// TwinCAT 3 PLC project CNM_CycleManager
// Title: CNM_CycleManager
// Company: ekvip automation GmbH
// Author: tdie
// ProjectVersion: 0.1.1.0
// Description: A library to provide Cycle management for use in simple state machines. .. <legal notes> legal notes ================= | SPDX-FileCopyrightText: © 2024 ekvip automation GmbH <info@ekvip.de> | SPDX-License-Identifier: Apache-2.0 | For details check: Apache-2.0_ .. _Apache-2.0: https://www.apache.org/licenses/LICENSE-2.0 .. </legal notes>
// ProgramVersion: 3.1.4026.19
// libraries:
//   CNM_AbstractObject, * (ekvip automation GmbH)
//   CNM_AssertionInterfaces, * (ekvip automation GmbH)
//   CNM_CommandInterfaces, * (ekvip automation GmbH)
//   CNM_CycleManagerInterfaces, * (ekvip automation GmbH)
//   CNM_MessageInterfaces, * (ekvip automation GmbH)
//   CNM_ReturnTypes, * (ekvip automation GmbH)
//   Tc2_Standard, * (Beckhoff Automation GmbH)
//   Tc2_System, * (Beckhoff Automation GmbH)
// project tree:
//   Commands/classes/ WaitCommand.TcPOU
//   Configurators/classes/ CycleManagerConfigurator.TcPOU, CycleManagerDefaultConfigurator.TcPOU, CycleManagerDefaultPausing.TcPOU, CycleManagerDefaultStepping.TcPOU, CycleManagerStepConfigurator.TcPOU, CycleManagerStepPausing.TcPOU, CycleManagerStepStepping.TcPOU
//   CycleManager/classes/ AbstractCycleManager.TcPOU, SimpleCycleManager.TcPOU
//   CycleManager/interfaces/ ICycleManagerStepParameters.TcIO
//   Project Information/ F_GetCompany.TcPOU, F_GetTitle.TcPOU, F_GetVersion.TcPOU
//   Version/ Global_Version.TcGVL

// ---- Version/Global_Version.TcGVL
{attribute 'TcGenerated'}
{attribute 'no-analysis'}
{attribute 'linkalways'}
// This function has been automatically generated from the project information.
VAR_GLOBAL CONSTANT
	{attribute 'const_non_replaced'}
	stLibVersion_CNM_CycleManager : ST_LibVersion := (iMajor := 0, iMinor := 1, iBuild := 1, iRevision := 0, nFlags := 0, sVersion := '0.1.1.0');
END_VAR

// ---- CycleManager/interfaces/ICycleManagerStepParameters.TcIO
(*

## Short summary
An interface to provide configurations for cycle manager steps.
Used internally to allow better fluent implementation.

.. <legal notes>

legal notes
=================
| SPDX-FileCopyrightText: © 2024 ekvip automation GmbH <info@ekvip.de>
| SPDX-License-Identifier: Apache-2.0
| For details check: Apache-2.0_

.. _Apache-2.0: https://www.apache.org/licenses/LICENSE-2.0

.. </legal notes>



*)
INTERFACE INTERNAL ICycleManagerStepParameters EXTENDS __System.IQueryInterface

PROPERTY currentErrorStep : DINT
SET
END_SET
END_PROPERTY

PROPERTY currentPauseEnabled : BOOL
SET
END_SET
END_PROPERTY

PROPERTY currentSteppingEnabled : BOOL
SET
END_SET
END_PROPERTY

PROPERTY currentStepWidth : DINT
SET
END_SET
END_PROPERTY

PROPERTY currentStopRequestMode :CNM_CycleManagerInterfaces.StepStopRequestMode
SET
END_SET
END_PROPERTY

PROPERTY currentTimeout : TIME
SET
END_SET
END_PROPERTY

PROPERTY currentTimeoutStep : DINT
SET
END_SET
END_PROPERTY

END_INTERFACE

// ---- Commands/classes/WaitCommand.TcPOU
(*

## Short summary
A simple command to wait for a given time.

.. <legal notes>

legal notes
=================
| SPDX-FileCopyrightText: © 2024 ekvip automation GmbH <info@ekvip.de>
| SPDX-License-Identifier: Apache-2.0
| For details check: Apache-2.0_

.. _Apache-2.0: https://www.apache.org/licenses/LICENSE-2.0

.. </legal notes>

*)
FUNCTION_BLOCK FINAL WaitCommand EXTENDS CNM_AbstractObject.Object IMPLEMENTS CNM_CommandInterfaces.ICommand
VAR
	timeToWait :TIME;
	timer :TON;
END_VAR

(*

## Short summary
This abstract property returns the class name of the concrete object, 
which is useful for logging/debugging purpose or to check the class name
for ``__DELETE`` in factories (sometimes it's necessary to do more 
than just to free the memory).

.. <legal notes>

legal notes
=================
| SPDX-FileCopyrightText: © 2022 ekvip automation GmbH <info@ekvip.de>
| SPDX-License-Identifier: Apache-2.0
| For details check: Apache-2.0_

.. _Apache-2.0: https://www.apache.org/licenses/LICENSE-2.0

.. </legal notes>

*)
PROPERTY className : CNM_AbstractObject.ClassName
GET
className := 'CNM_CycleManager.WaitCommand';
END_GET
END_PROPERTY

(*

## Short summary
Executes the action associated with this command.

.. <legal notes>

legal notes
=================
| SPDX-FileCopyrightText: © 2022 ekvip automation GmbH <info@ekvip.de>
| SPDX-License-Identifier: Apache-2.0
| For details check: Apache-2.0_

.. _Apache-2.0: https://www.apache.org/licenses/LICENSE-2.0

.. </legal notes>

*)
METHOD executeCommand : CNM_ReturnTypes.SingleExecutionState
VAR_INPUT
	(*control bit to start or abort the command*)
	execute	: BOOL;
END_VAR
THIS^.timer(IN := execute AND (THIS^.waitTime <> T#0S), PT := THIS^.waitTime);
IF(THIS^.timer.Q OR_ELSE THIS^.waitTime = T#0S)THEN
	executeCommand := CNM_ReturnTypes.SingleExecutionState.SUCCESS;
ELSE
	executeCommand := CNM_ReturnTypes.SingleExecutionState.BUSY;	
END_IF
END_METHOD

(*

## Short summary
The constructor ``FB_init`` is needed to create an unique hash code.
The hash code is a pseudo random number create with a xorshift_ algorithm.
It can be overwritten on derivations, because it will be called implicit, ``SUPER^.FB_init()`` is not required.
For more information check: `Behavoir with derived function blocks`_

.. _Behavoir with derived function blocks: https://infosys.beckhoff.com/content/1033/tc3_plc_intro/5482088715.html?id=6983869892358031022
.. _xorshift: https://en.wikipedia.org/wiki/Xorshift

.. <legal notes>

legal notes
=================
| SPDX-FileCopyrightText: © 2022 ekvip automation GmbH <info@ekvip.de>
| SPDX-License-Identifier: Apache-2.0
| For details check: Apache-2.0_

.. _Apache-2.0: https://www.apache.org/licenses/LICENSE-2.0

.. </legal notes>

*)
METHOD FB_init :BOOL
VAR_INPUT
	(* if TRUE, the retain variables are initialized (warm start / cold start)*)
	bInitRetains	:BOOL;
	(* if TRUE, the instance afterwards gets moved into the copy code (online change) *)
	bInCopyCode	:BOOL;
	(* time to wait until return state is success *)
	waitTime :TIME;
END_VAR
THIS^.timeToWait := waitTime;
END_METHOD

(*

## Short summary
This property sets or gets the time to wait for until the command returns SUCCESS.

.. <legal notes>

legal notes
=================
| SPDX-FileCopyrightText: © 2022 ekvip automation GmbH <info@ekvip.de>
| SPDX-License-Identifier: Apache-2.0
| For details check: Apache-2.0_

.. _Apache-2.0: https://www.apache.org/licenses/LICENSE-2.0

.. </legal notes>

*)
PROPERTY waitTime : TIME
GET
waitTime := THIS^.timeToWait;
END_GET
SET
THIS^.timeToWait := waitTime;
END_SET
END_PROPERTY

END_FUNCTION_BLOCK

// ---- Configurators/classes/CycleManagerConfigurator.TcPOU
(*

## Short summary
A class to provide fluent access to the configuration scope of a cycle manager.

.. <legal notes>

legal notes
=================
| SPDX-FileCopyrightText: © 2024 ekvip automation GmbH <info@ekvip.de>
| SPDX-License-Identifier: Apache-2.0
| For details check: Apache-2.0_

.. _Apache-2.0: https://www.apache.org/licenses/LICENSE-2.0

.. </legal notes>



*)
FUNCTION_BLOCK INTERNAL CycleManagerConfigurator IMPLEMENTS CNM_CycleManagerInterfaces.ICycleManagerConfigurationScope
VAR
	cycleManagerDefault :CNM_CycleManagerInterfaces.ICycleManagerDefaultParameters;
	cycleManagerStep :ICycleManagerStepParameters;
	stepConfigurator :CycleManagerStepConfigurator();
	defaultConfigurator :CycleManagerDefaultConfigurator();
END_VAR

(*

## Short summary
Initializes the CycleManagerConfigurator with required cycle manager parameters.

.. <legal notes>

legal notes
=================
| SPDX-FileCopyrightText: © 2025 ekvip automation GmbH <info@ekvip.de>
| SPDX-License-Identifier: Apache-2.0
| For details check: Apache-2.0_

.. _Apache-2.0: https://www.apache.org/licenses/LICENSE-2.0

.. </legal notes>

*)
//FB_Init is always available implicitly and it is used primarily for initialization.
//The return value is not evaluated. For a specific influence, you can also declare the
//methods explicitly and provide additional code there with the standard initialization
//code. You can evaluate the return value.
METHOD FB_Init: BOOL
VAR_INPUT
    bInitRetains: BOOL; // TRUE: the retain variables are initialized (reset warm / reset cold)
    bInCopyCode: BOOL;  // TRUE: the instance will be copied to the copy code afterward (online change)   
	cycleManagerDefault :CNM_CycleManagerInterfaces.ICycleManagerDefaultParameters; //Interface for default cycle manager parameters
	cycleManagerStep :ICycleManagerStepParameters; //Interface for step-specific cycle manager parameters
END_VAR
THIS^.cycleManagerDefault := cycleManagerDefault;
THIS^.cycleManagerStep := cycleManagerStep;
THIS^.defaultConfigurator.cycleManager := cycleManagerDefault;
THIS^.stepConfigurator.cycleManager := cycleManagerStep;
END_METHOD

(*

## Short summary
Provides access to sequence-level configuration for all cycle manager steps.

### Purpose and usage
This property returns the sequence configuration interface that allows setting default parameters
for all steps in the cycle manager. It provides a fluent interface for configuring sequence-wide
settings that apply to the entire cycle execution.

The sequence configuration affects all steps uniformly and provides default values for:
- Pause behavior
- Stepping mode settings
- Stop request handling
- Other sequence-wide parameters


### typical usage patterns
1. **Setting default timeouts**: Configure default timeout for all steps
2. **Pause configuration**: Set pause behavior for the entire sequence
3. **Stepping mode**: Configure stepping mode defaults
4. **Stop handling**: Define how stop requests are handled globally

### When to use
- When you need to configure default behavior for all steps
- To set sequence-wide parameters that apply uniformly
- For configuring global cycle manager behavior
- When implementing consistent behavior across all steps

### Example
```
// Configure sequence defaults
cycleManager.configuration.configuration.sequence
    .pauseConfiguration
        .pauseAllowed(TRUE)
        .pauseTimeout(T#5S);

// Set stepping mode for entire sequence
cycleManager.configuration.configuration.sequence
    .steppingConfiguration
        .steppingEnabled(debugMode)
        .autoStepDelay(T#100MS);

// Configure stop request handling
cycleManager.configuration.configuration.sequence
    .stopRequestConfiguration
        .stopAllowed(TRUE)
        .immediateStop(FALSE);

```
.. <legal notes>

legal notes
=================
| SPDX-FileCopyrightText: © 2025 ekvip automation GmbH <info@ekvip.de>
| SPDX-License-Identifier: Apache-2.0
| For details check: Apache-2.0_

.. _Apache-2.0: https://www.apache.org/licenses/LICENSE-2.0

.. </legal notes>

*)
PROPERTY sequence : CNM_CycleManagerInterfaces.ISequenceConfiguration
GET
sequence := defaultConfigurator;
END_GET
END_PROPERTY

(*

## Short summary
Provides access to step-specific configuration for individual cycle manager steps.

### Purpose and usage
This property returns the step configuration interface that allows setting parameters
for specific steps in the cycle manager. It provides a fluent interface for configuring
individual step behavior that overrides the sequence defaults.

The step configuration allows fine-grained control over individual steps including:
- Step-specific timeouts
- Individual pause behavior
- Custom stepping settings
- Step-specific stop handling

### typical usage patterns
1. **Step-specific timeouts**: Override default timeout for critical steps
2. **Disable pause**: Prevent pausing on critical operation steps
3. **Skip stepping**: Make certain steps non-steppable in debug mode
4. **Custom behavior**: Define unique behavior for specific steps

### When to use
- When specific steps need different behavior than the sequence default
- For critical steps that should not be pausable or steppable
- To set custom timeouts for long-running operations
- When implementing step-specific error handling

### Example
```
// Configure specific step with custom timeout
cycleManager.configuration.configuration.step
    .forStep(MySteps.LONG_OPERATION)
    .setTimeout(T#30S)
    .pauseAllowed(FALSE);  // Critical step - no pause allowed

// Configure multiple steps
cycleManager.configuration.configuration.step
    .forStep(MySteps.INIT)
    .setTimeout(T#5S)
    .steppingAllowed(TRUE);

cycleManager.configuration.configuration.step
    .forStep(MySteps.CRITICAL_PROCESS)
    .setTimeout(T#10S)
    .pauseAllowed(FALSE)
    .stopAllowed(FALSE);  // Must complete once started

// Configure error step
cycleManager.configuration.configuration.step
    .forStep(DefaultSteps.STEP.ERROR)
    .setTimeout(T#0S)  // No timeout in error state
    .steppingAllowed(TRUE);  // Allow stepping through error handling
```

.. <legal notes>

legal notes
=================
| SPDX-FileCopyrightText: © 2025 ekvip automation GmbH <info@ekvip.de>
| SPDX-License-Identifier: Apache-2.0
| For details check: Apache-2.0_

.. _Apache-2.0: https://www.apache.org/licenses/LICENSE-2.0

.. </legal notes>


*)
PROPERTY step : CNM_CycleManagerInterfaces.IStepConfiguration
GET
VAR_INST
	conf :CycleManagerStepConfigurator();
END_VAR
step := stepConfigurator;
END_GET
END_PROPERTY

END_FUNCTION_BLOCK

// ---- Configurators/classes/CycleManagerStepConfigurator.TcPOU
(*

## Short summary
A class to provide fluent access to the current step configuration of a cycle manager.

.. <legal notes>

legal notes
=================
| SPDX-FileCopyrightText: © 2024 ekvip automation GmbH <info@ekvip.de>
| SPDX-License-Identifier: Apache-2.0
| For details check: Apache-2.0_

.. _Apache-2.0: https://www.apache.org/licenses/LICENSE-2.0

.. </legal notes>



*)
FUNCTION_BLOCK INTERNAL CycleManagerStepConfigurator IMPLEMENTS CNM_CycleManagerInterfaces.IStepConfiguration, CNM_CycleManagerInterfaces.IStopRequestConfiguration
VAR
	parameters :ICycleManagerStepParameters;
	pauserator :CycleManagerStepPausing();
	steperator :CycleManagerStepStepping();
END_VAR

(*

## Short summary
Sets the stop request behavior to execute after successful step completion for the current step.

### Purpose and usage
This method configures the current step to process stop requests only after the step has completed successfully.
This setting overrides the sequence default for this specific step. When this mode is active, stop requests
received during step execution will be deferred until the step completes with success.

This ensures that the specific step completes successfully before the cycle is stopped,
maintaining data integrity and process consistency for critical operations.

### typical usage patterns
1. **Critical steps**: Ensure specific steps complete before stopping
2. **Transaction steps**: Finish data transactions cleanly
3. **Safety operations**: Complete safety-critical steps
4. **Production steps**: Avoid partial operations on key steps

### When to use
- For steps that must complete successfully before stopping
- When specific operations should not be interrupted
- For data consistency in critical steps
- To override sequence defaults for important steps

### Example
```
// Configure specific step for safe stopping
cycleManager.configuration.configuration.step
    .stopRequest
    .afterSuccess();

// Apply to critical step during configuration
CASE cycleManager.steps.current OF
    MySteps.INIT:
        // Configure next critical step
        cycleManager.configuration.configuration.step
            .timeout := T#10S;
        cycleManager.configuration.configuration.step
            .stopRequest.afterSuccess();
        cycleManager.steps.next := MySteps.CRITICAL_WRITE;
        
    MySteps.CRITICAL_WRITE:
        // This step will complete before stop is processed
        IF writeCriticalData() THEN
            cycleManager.steps.next := MySteps.NEXT_STEP;
        END_IF;
END_CASE
```


.. <legal notes>

legal notes
=================
| SPDX-FileCopyrightText: © 2025 ekvip automation GmbH <info@ekvip.de>
| SPDX-License-Identifier: Apache-2.0
| For details check: Apache-2.0_

.. _Apache-2.0: https://www.apache.org/licenses/LICENSE-2.0

.. </legal notes>

*)
METHOD afterSuccessfulStep
THIS^.cycleManager.currentStopRequestMode := CNM_CycleManagerInterfaces.StepStopRequestMode.AFTER_SUCCESSFUL_STEP;
END_METHOD

(*

## Short summary
Gets or sets the cycle manager step parameters interface used by this configurator.

### Purpose and usage
This property provides access to the underlying cycle manager step parameters interface.
It allows getting the current cycle manager instance and setting a new one if needed.

When setting a new cycle manager, all internal configurators (stepping and pausing)
are automatically updated to use the new instance. This property manages step-specific
parameters that override sequence defaults.

### typical usage patterns
1. **Initialization**: Set during configurator creation
2. **Runtime changes**: Switch cycle manager instances
3. **Access parameters**: Get current cycle manager for direct access
4. **Step-specific config**: Access step-level parameters

### When to use
- During initialization to set the cycle manager
- When switching between different cycle manager implementations
- For direct access to step-specific parameters
- In factory patterns for dynamic configuration

### Example
```
// Get current cycle manager
VAR
    currentManager : ICycleManagerStepParameters;
END_VAR

currentManager := stepConfigurator.cycleManager;

// Set new cycle manager
VAR
    newManager : MyCycleManagerStepImplementation;
END_VAR

stepConfigurator.cycleManager := newManager;
// All sub-configurators now use newManager

// Direct parameter access
IF stepConfigurator.cycleManager.currentTimeout > T#5S THEN
    // Handle long timeout for current step
END_IF;
```

.. <legal notes>

legal notes
=================
| SPDX-FileCopyrightText: © 2025 ekvip automation GmbH <info@ekvip.de>
| SPDX-License-Identifier: Apache-2.0
| For details check: Apache-2.0_

.. _Apache-2.0: https://www.apache.org/licenses/LICENSE-2.0

.. </legal notes>


*)
PROPERTY cycleManager : ICycleManagerStepParameters
GET
cycleManager := THIS^.parameters;
END_GET
SET
THIS^.parameters := cycleManager;
THIS^.steperator.cycleManager := THIS^.cycleManager;
THIS^.pauserator.cycleManager := THIS^.cycleManager;
END_SET
END_PROPERTY

(*

## Short summary
This property sets the next step in case of an error.
Is reset to the default ERROR_STEP when the current step changes.

.. <legal notes>

legal notes
=================
| SPDX-FileCopyrightText: © 2024 ekvip automation GmbH <info@ekvip.de>
| SPDX-License-Identifier: Apache-2.0
| For details check: Apache-2.0_

.. _Apache-2.0: https://www.apache.org/licenses/LICENSE-2.0

.. </legal notes>

*)
PROPERTY errorStep : DINT
SET
THIS^.cycleManager.currentErrorStep := errorStep;
END_SET
END_PROPERTY

(*

## Short summary
Initializes the CycleManagerStepConfigurator and its sub-configurators.

.. <legal notes>

legal notes
=================
| SPDX-FileCopyrightText: © 2025 ekvip automation GmbH <info@ekvip.de>
| SPDX-License-Identifier: Apache-2.0
| For details check: Apache-2.0_

.. _Apache-2.0: https://www.apache.org/licenses/LICENSE-2.0

.. </legal notes>

*)
//FB_Init is always available implicitly and it is used primarily for initialization.
//The return value is not evaluated. For a specific influence, you can also declare the
//methods explicitly and provide additional code there with the standard initialization
//code. You can evaluate the return value.
METHOD FB_Init: BOOL
VAR_INPUT
    bInitRetains: BOOL; // TRUE: the retain variables are initialized (reset warm / reset cold)
    bInCopyCode: BOOL;  // TRUE: the instance will be copied to the copy code afterward (online change)   
END_VAR
THIS^.steperator.cycleManager := THIS^.cycleManager;
THIS^.pauserator.cycleManager := THIS^.cycleManager;
END_METHOD

(*

## Short summary
Sets the stop request behavior to ignore all stop requests for the current step.

### Purpose and usage
This method configures the current step to completely ignore all stop requests.
This setting overrides the sequence default for this specific step. When this mode
is active, stop requests will not be processed at all during this step, and the
step will continue running until completion or error.

This mode should be used with extreme caution as it prevents normal stopping
mechanisms from working for the specific step.

### typical usage patterns
1. **Atomic operations**: Steps that must complete without interruption
2. **Safety sequences**: Emergency procedures for specific steps
3. **Critical writes**: Database or file operations that cannot be stopped
4. **Hardware operations**: Steps controlling physical processes

### When to use
- For step-specific critical operations that must complete
- During safety-critical step sequences
- For atomic operations within a larger sequence
- When a specific step must ignore stop requests
- Use with extreme caution - limits operator control

### Example
```
// Configure specific step to ignore stops
cycleManager.configuration.configuration.step
    .stopRequest
    .ignore();

// Apply to critical hardware operation
CASE cycleManager.steps.current OF
    MySteps.PREPARE_CRITICAL:
        // Configure next step to ignore stops
        cycleManager.configuration.configuration.step
            .stopRequest.ignore();
        cycleManager.steps.next := MySteps.CRITICAL_HARDWARE_OP;
        
    MySteps.CRITICAL_HARDWARE_OP:
        // This step ignores all stop requests
        IF performCriticalHardwareOperation() THEN
            // Re-enable stop handling for next step
            cycleManager.configuration.configuration.step
                .stopRequest.afterSuccess();
            cycleManager.steps.next := MySteps.NORMAL_OPERATION;
        END_IF;
END_CASE

// Stop requests during critical step will be ignored
IF stopButton THEN
    cycleManager.requestStop();  // No effect on CRITICAL_HARDWARE_OP
END_IF;
```

.. <legal notes>

legal notes
=================
| SPDX-FileCopyrightText: © 2025 ekvip automation GmbH <info@ekvip.de>
| SPDX-License-Identifier: Apache-2.0
| For details check: Apache-2.0_

.. _Apache-2.0: https://www.apache.org/licenses/LICENSE-2.0

.. </legal notes>


*)
METHOD ignore
THIS^.cycleManager.currentStopRequestMode := CNM_CycleManagerInterfaces.StepStopRequestMode.IGNORE;
END_METHOD

(*

## Short summary
Sets the stop request behavior to always process stop requests immediately for the current step.

### Purpose and usage
This method configures the current step to always process stop requests immediately,
regardless of the step's execution state or outcome. This setting overrides the sequence
default for this specific step. Stop requests are handled as soon as they are received,
potentially interrupting the current operation.

This mode provides the most responsive stop behavior for the specific step but may
interrupt operations that are in progress.

### typical usage patterns
1. **Non-critical steps**: Allow immediate stop on safe steps
2. **Wait steps**: Enable quick response during waits
3. **User interaction**: Responsive stops during user steps
4. **Idle states**: Allow immediate stop when idle

### When to use
- For steps where immediate stop response is acceptable
- During wait or idle steps
- For non-critical operations that can be interrupted
- To override restrictive sequence defaults for specific steps

### Example
```
// Configure specific step for immediate stop
cycleManager.configuration.configuration.step
    .stopRequest
    .always();

// Apply to wait steps
CASE cycleManager.steps.current OF
    MySteps.WAIT_FOR_INPUT:
        // This step can be interrupted immediately
        cycleManager.configuration.configuration.step
            .stopRequest.always();
        IF inputReceived THEN
            cycleManager.steps.next := MySteps.PROCESS_INPUT;
        END_IF;
        
    MySteps.IDLE:
        // Idle step allows immediate stop
        cycleManager.configuration.configuration.step
            .stopRequest.always();
        IF startCommand THEN
            cycleManager.steps.next := MySteps.START_PROCESS;
        END_IF;
END_CASE
```

.. <legal notes>

legal notes
=================
| SPDX-FileCopyrightText: © 2025 ekvip automation GmbH <info@ekvip.de>
| SPDX-License-Identifier: Apache-2.0
| For details check: Apache-2.0_

.. _Apache-2.0: https://www.apache.org/licenses/LICENSE-2.0

.. </legal notes>

*)
METHOD immediate
THIS^.cycleManager.currentStopRequestMode := CNM_CycleManagerInterfaces.StepStopRequestMode.IMMEDIATE;
END_METHOD

(*

## Short summary
This method sets the stop request behaviour to ``StepStopRequestMode.AFTER_NOT_SUCCESS``.

.. <legal notes>

legal notes
=================
| SPDX-FileCopyrightText: © 2024 ekvip automation GmbH <info@ekvip.de>
| SPDX-License-Identifier: Apache-2.0
| For details check: Apache-2.0_

.. _Apache-2.0: https://www.apache.org/licenses/LICENSE-2.0

.. </legal notes>

*)
METHOD onBusy
THIS^.cycleManager.currentStopRequestMode := CNM_CycleManagerInterfaces.StepStopRequestMode.ON_BUSY;
END_METHOD

(*

## Short summary
Provides access to the pause configuration for the current cycle manager step.

### Purpose and usage
This property returns the pause configuration interface that allows setting pause-related
parameters for the current step. It provides a fluent interface for configuring how
the cycle manager handles pause requests for this specific step, overriding sequence defaults.

The pause configuration controls:
- Whether pausing is allowed for this step
- Step-specific pause timeout behavior
- Resume conditions for this step
- Step-specific pause state handling


### typical usage patterns
1. **Disable pause**: Prevent pausing on critical steps
2. **Enable pause**: Allow pausing on safe steps
3. **Override defaults**: Change pause behavior for specific steps
4. **Step-specific timeout**: Set different pause timeout for steps

### When to use
- To prevent pausing during critical operations
- To enable pausing on specific wait or idle steps
- When step-specific pause behavior differs from sequence default
- For fine-grained pause control in complex sequences

### Example
```
// Disable pause for critical step
CASE cycleManager.steps.current OF
    MySteps.PREPARE_CRITICAL:
        cycleManager.configuration.configuration.step
            .pause.disable();
        cycleManager.steps.next := MySteps.CRITICAL_OPERATION;
        
    MySteps.WAIT_FOR_USER:
        // Enable pause for wait step
        cycleManager.configuration.configuration.step
            .pause.enable();
        IF userInput THEN
            cycleManager.steps.next := MySteps.PROCESS_INPUT;
        END_IF;
END_CASE

// Configure step with specific pause settings
cycleManager.configuration.configuration.step
    .pause
    .enable()
    .timeout(T#60S);  // Longer pause allowed for this step

```

.. <legal notes>

legal notes
=================
| SPDX-FileCopyrightText: © 2025 ekvip automation GmbH <info@ekvip.de>
| SPDX-License-Identifier: Apache-2.0
| For details check: Apache-2.0_

.. _Apache-2.0: https://www.apache.org/licenses/LICENSE-2.0

.. </legal notes>

*)
PROPERTY pause : CNM_CycleManagerInterfaces.IPauseConfiguration
GET
VAR_INST
END_VAR
pause := pauserator;
END_GET
END_PROPERTY

(*

## Short summary
Provides access to the stepping configuration for the current cycle manager step.

### Purpose and usage
This property returns the stepping configuration interface that allows setting stepping-related
parameters for the current step. It provides a fluent interface for configuring step-by-step
execution mode for this specific step, overriding sequence defaults.

The stepping configuration controls:
- Whether stepping mode is enabled for this step
- Step-specific auto-step delays
- Step trigger conditions
- Single-step behavior for this step


### typical usage patterns
1. **Skip stepping**: Disable stepping for automated steps
2. **Force stepping**: Require manual confirmation for critical steps
3. **Custom delays**: Set step-specific auto-step timing
4. **Debug control**: Enable stepping only for complex steps

### When to use
- To skip stepping mode for simple or automated steps
- To force stepping on critical steps even in auto mode
- When specific steps need different stepping behavior
- For debugging specific steps in a sequence

### Example
```
// Disable stepping for automated steps
CASE cycleManager.steps.current OF
    MySteps.AUTO_CALCULATION:
        // This step runs without stepping even in debug mode
        cycleManager.configuration.configuration.step
            .stepping.disable();
        performCalculations();
        cycleManager.steps.next := MySteps.VERIFY_RESULTS;
        
    MySteps.VERIFY_RESULTS:
        // Force stepping for verification
        cycleManager.configuration.configuration.step
            .stepping.enable();
        IF resultsValid THEN
            cycleManager.steps.next := MySteps.CONTINUE;
        END_IF;
END_CASE

// Configure step with specific stepping settings
cycleManager.configuration.configuration.step
    .stepping
    .enable()
    .autoStep(TRUE)
    .autoStepDelay(T#5S);  // Slower auto-step for this step
```

.. <legal notes>

legal notes
=================
| SPDX-FileCopyrightText: © 2025 ekvip automation GmbH <info@ekvip.de>
| SPDX-License-Identifier: Apache-2.0
| For details check: Apache-2.0_

.. _Apache-2.0: https://www.apache.org/licenses/LICENSE-2.0

.. </legal notes>

*)
PROPERTY stepping : CNM_CycleManagerInterfaces.ISteppingConfiguration
GET
stepping := steperator;
END_GET
END_PROPERTY

(*

## Short summary
Sets the step width for automatic step increment for the current step.

### Purpose and usage
This property sets the increment value used when automatically advancing from the current step.
It overrides the sequence default step width for this specific step. When no explicit next step
is specified, the cycle manager will advance by this step width value.

This allows individual steps to have different increment values, useful for:
- Skipping blocks of steps
- Jumping to different sequence sections
- Implementing conditional branching
- Custom step numbering schemes

### typical usage patterns
1. **Skip sections**: Large step width to jump over optional sections
2. **Branch control**: Different widths for different branches
3. **Return jumps**: Negative values to go back in sequence
4. **Custom flow**: Implement complex sequencing logic

### When to use
- When this step needs to jump to a non-sequential next step
- For implementing branching logic
- To skip optional sequence sections
- When overriding the default sequential flow

### Example
```
// Configure step to skip optional section
CASE cycleManager.steps.current OF
    100:  // Decision step
        IF skipOptionalSteps THEN
            // Jump to step 200, skipping 110-190
            cycleManager.configuration.configuration.step
                .stepWidth := 100;
        ELSE
            // Normal increment to 110
            cycleManager.configuration.configuration.step
                .stepWidth := 10;
        END_IF;
        cycleManager.steps.next := 0;  // Use automatic increment
        
    190:  // Last optional step
        // Ensure we continue at 200
        cycleManager.configuration.configuration.step
            .stepWidth := 10;
        cycleManager.steps.next := 0;  // Automatically goes to 200
        
    250:  // Loop back step
        IF repeatRequired THEN
            // Go back to step 200
            cycleManager.configuration.configuration.step
                .stepWidth := -50;
            cycleManager.steps.next := 0;  // Automatically goes to 200
        END_IF;
END_CASE
```

.. <legal notes>

legal notes
=================
| SPDX-FileCopyrightText: © 2025 ekvip automation GmbH <info@ekvip.de>
| SPDX-License-Identifier: Apache-2.0
| For details check: Apache-2.0_

.. _Apache-2.0: https://www.apache.org/licenses/LICENSE-2.0

.. </legal notes>

*)
PROPERTY stepWidth : DINT
SET
THIS^.cycleManager.currentStepWidth := stepWidth;
END_SET
END_PROPERTY

(*

## Short summary
Provides access to the stop request configuration interface for the current step.

### Purpose and usage
This property returns the stop request configuration interface for the current step,
providing access to methods that configure how the cycle manager handles stop requests
for this specific step. The configurator itself implements the IStopRequestConfiguration interface.

This allows step-specific stop behavior that overrides sequence defaults:
- always(): Process stop requests immediately for this step
- afterSuccess(): Process after this step completes successfully
- afterNotSuccess(): Process after this step fails
- ignore(): Ignore all stop requests for this step


### typical usage patterns
1. **Critical steps**: Configure to ignore or defer stops
2. **Safe steps**: Allow immediate stop processing
3. **Conditional stops**: Different behavior based on step outcome
4. **Override defaults**: Step-specific stop handling

### When to use
- To customize stop behavior for specific steps
- When certain steps need different stop handling than the sequence default
- For implementing step-specific safety requirements
- To ensure critical steps complete before stopping

### Example
```
// Configure critical step to complete before stop
CASE cycleManager.steps.current OF
    MySteps.PREPARE_CRITICAL:
        cycleManager.configuration.configuration.step
            .stopRequest.afterSuccess();
        cycleManager.steps.next := MySteps.CRITICAL_WRITE;
        
    MySteps.WAIT_STEP:
        // Allow immediate stop during wait
        cycleManager.configuration.configuration.step
            .stopRequest.always();
        IF condition THEN
            cycleManager.steps.next := MySteps.CONTINUE;
        END_IF;
        
    MySteps.ATOMIC_OPERATION:
        // This step cannot be stopped
        cycleManager.configuration.configuration.step
            .stopRequest.ignore();
        performAtomicOperation();
        cycleManager.steps.next := MySteps.NEXT;
END_CASE

// Chain with other step configurations
cycleManager.configuration.configuration.step
    .timeout := T#5S;
    .stopRequest.afterSuccess();
    .pause.disable();

```

.. <legal notes>

legal notes
=================
| SPDX-FileCopyrightText: © 2025 ekvip automation GmbH <info@ekvip.de>
| SPDX-License-Identifier: Apache-2.0
| For details check: Apache-2.0_

.. _Apache-2.0: https://www.apache.org/licenses/LICENSE-2.0

.. </legal notes>


*)
PROPERTY stopRequest : CNM_CycleManagerInterfaces.IStopRequestConfiguration
GET
stopRequest := THIS^;
END_GET
END_PROPERTY

(*

## Short summary
This property sets the maximum execution time for the current step. 
The cycle manager will go into the error step after the time elapsed.
Set to T#0MS for no timeout.

.. <legal notes>

legal notes
=================
| SPDX-FileCopyrightText: © 2024 ekvip automation GmbH <info@ekvip.de>
| SPDX-License-Identifier: Apache-2.0
| For details check: Apache-2.0_

.. _Apache-2.0: https://www.apache.org/licenses/LICENSE-2.0

.. </legal notes>

*)
PROPERTY timeout : TIME
SET
THIS^.cycleManager.currentTimeout := timeout;
END_SET
END_PROPERTY

(*

## Short summary
This property sets the step that will be set if the current step reaches a timeout. 
Will by default be the error step and reset after the current step changes.

.. <legal notes>

legal notes
=================
| SPDX-FileCopyrightText: © 2024 ekvip automation GmbH <info@ekvip.de>
| SPDX-License-Identifier: Apache-2.0
| For details check: Apache-2.0_

.. _Apache-2.0: https://www.apache.org/licenses/LICENSE-2.0

.. </legal notes>

*)
PROPERTY timeoutStep : DINT
SET
THIS^.cycleManager.currentTimeoutStep := timeoutStep;
END_SET
END_PROPERTY

END_FUNCTION_BLOCK

// ---- Configurators/classes/CycleManagerStepPausing.TcPOU
(*

## Short summary
A class to provide fluent access to the current step pause configuration of a cycle manager.

.. <legal notes>

legal notes
=================
| SPDX-FileCopyrightText: © 2024 ekvip automation GmbH <info@ekvip.de>
| SPDX-License-Identifier: Apache-2.0
| For details check: Apache-2.0_

.. _Apache-2.0: https://www.apache.org/licenses/LICENSE-2.0

.. </legal notes>



*)
FUNCTION_BLOCK INTERNAL CycleManagerStepPausing IMPLEMENTS CNM_CycleManagerInterfaces.IPauseConfiguration
VAR
	parameters :ICycleManagerStepParameters;
END_VAR

(*

## Short summary
Gets or sets the cycle manager step parameters interface used for pause configuration.

### Purpose and usage
This property provides access to the underlying cycle manager step parameters interface
that this pause configurator operates on. It allows getting the current cycle manager instance
and setting a new one if needed for step-specific pause configuration.

The property is primarily used internally but can be accessed for direct parameter manipulation
or when switching between different cycle manager instances at the step level.

### typical usage patterns
1. **Internal initialization**: Set during configurator setup
2. **Runtime switching**: Change cycle manager instances
3. **Direct access**: Get parameters for advanced step configuration
4. **Dependency injection**: Inject different implementations

### When to use
- During initialization to connect to a cycle manager
- When switching between different cycle manager implementations
- For direct access to step-specific pause parameters
- In advanced configuration scenarios for individual steps

### Example
```
// Get current cycle manager
VAR
    currentManager : ICycleManagerStepParameters;
END_VAR

currentManager := stepPauseConfig.cycleManager;

// Check current step pause state
IF currentManager.currentPauseEnabled THEN
    // Pause is enabled for current step
END_IF;

// Set new cycle manager
VAR
    newManager : MyCycleManagerStepImplementation;
END_VAR

stepPauseConfig.cycleManager := newManager;
```

.. <legal notes>

legal notes
=================
| SPDX-FileCopyrightText: © 2025 ekvip automation GmbH <info@ekvip.de>
| SPDX-License-Identifier: Apache-2.0
| For details check: Apache-2.0_

.. _Apache-2.0: https://www.apache.org/licenses/LICENSE-2.0

.. </legal notes>

*)
PROPERTY cycleManager : ICycleManagerStepParameters
GET
cycleManager := THIS^.parameters;
END_GET
SET
THIS^.parameters := cycleManager;
END_SET
END_PROPERTY

(*

## Short summary
Disables pause functionality for the current cycle manager step.

### Purpose and usage
This method disables the pause functionality for the current step only, overriding
the sequence default. When pause is disabled for a step, pause requests will be
ignored while this step is executing, ensuring the step runs to completion.

Disabling pause at the step level is useful for:
- Critical operations within a pausable sequence
- Time-sensitive steps that must not be interrupted
- Atomic operations that need to complete
- Safety-critical step procedures

### typical usage patterns
1. **Critical steps**: Prevent pausing during important operations
2. **Time-sensitive**: Steps with timing requirements
3. **Atomic operations**: Multi-part steps that must complete together
4. **Override sequence**: Disable pause for specific steps only

### When to use
- For steps that must complete without interruption
- During critical operations within a larger sequence
- For time-sensitive or atomic step operations
- When specific steps should override sequence pause settings

### Example
```
// Disable pause for critical step
CASE cycleManager.steps.current OF
    MySteps.PREPARE_CRITICAL:
        // Next step cannot be paused
        cycleManager.configuration.configuration.step
            .pause.disable();
        cycleManager.steps.next := MySteps.CRITICAL_WRITE;
        
    MySteps.CRITICAL_WRITE:
        // This step runs without pause possibility
        IF writeCriticalData() THEN
            // Re-enable pause for next step
            cycleManager.configuration.configuration.step
                .pause.enable();
            cycleManager.steps.next := MySteps.NORMAL_OPERATION;
        END_IF;
END_CASE

// Temporarily disable pause for atomic operation
IF startAtomicOperation THEN
    cycleManager.configuration.configuration.step
        .pause.disable();
    cycleManager.configuration.configuration.step
        .timeout := T#30S;  // Ensure completion
END_IF;
```

.. <legal notes>

legal notes
=================
| SPDX-FileCopyrightText: © 2025 ekvip automation GmbH <info@ekvip.de>
| SPDX-License-Identifier: Apache-2.0
| For details check: Apache-2.0_

.. _Apache-2.0: https://www.apache.org/licenses/LICENSE-2.0

.. </legal notes>

*)
METHOD disable
THIS^.cycleManager.currentPauseEnabled := FALSE;
END_METHOD

(*

## Short summary
Enables pause functionality for the current cycle manager step.

### Purpose and usage
This method enables the pause functionality for the current step only, overriding
the sequence default if necessary. When pause is enabled for a step, the cycle
can be paused while this step is executing, allowing operators to halt execution.

Enabling pause at the step level is useful for:
- Wait or idle steps where pausing is safe
- User interaction steps
- Steps where operator inspection may be needed
- Override sequence settings for specific steps

### typical usage patterns
1. **Wait steps**: Enable pause during wait operations
2. **User steps**: Allow pause during user interactions
3. **Inspection points**: Enable pause for quality checks
4. **Override sequence**: Enable pause for specific steps only

### When to use
- For steps where pausing is safe and desired
- During wait or idle operations
- At inspection or decision points in the sequence
- When specific steps should allow pausing regardless of sequence settings

### Example
```
// Enable pause for wait step
CASE cycleManager.steps.current OF
    MySteps.WAIT_FOR_OPERATOR:
        // This step can be paused
        cycleManager.configuration.configuration.step
            .pause.enable();
        IF operatorReady THEN
            cycleManager.steps.next := MySteps.CONTINUE;
        END_IF;
        
    MySteps.INSPECTION_POINT:
        // Enable pause for inspection
        cycleManager.configuration.configuration.step
            .pause.enable();
        cycleManager.configuration.configuration.step
            .timeout := T#0S;  // No timeout during inspection
        IF inspectionComplete THEN
            cycleManager.steps.next := MySteps.NEXT;
        END_IF;
END_CASE

// Conditionally enable pause
IF debugMode OR maintenanceMode THEN
    cycleManager.configuration.configuration.step
        .pause.enable();
END_IF;

// Handle pause request for enabled step
IF cycleManager.currentPauseEnabled AND pauseRequested THEN
    cycleManager.requestPause();
END_IF;
```

.. <legal notes>

legal notes
=================
| SPDX-FileCopyrightText: © 2025 ekvip automation GmbH <info@ekvip.de>
| SPDX-License-Identifier: Apache-2.0
| For details check: Apache-2.0_

.. _Apache-2.0: https://www.apache.org/licenses/LICENSE-2.0

.. </legal notes>

*)
METHOD enable
THIS^.cycleManager.currentPauseEnabled := TRUE;
END_METHOD

END_FUNCTION_BLOCK

// ---- Configurators/classes/CycleManagerStepStepping.TcPOU
(*

## Short summary
A class to provide fluent access to the current step stepping configuration of a cycle manager.

.. <legal notes>

legal notes
=================
| SPDX-FileCopyrightText: © 2024 ekvip automation GmbH <info@ekvip.de>
| SPDX-License-Identifier: Apache-2.0
| For details check: Apache-2.0_

.. _Apache-2.0: https://www.apache.org/licenses/LICENSE-2.0

.. </legal notes>



*)
FUNCTION_BLOCK INTERNAL CycleManagerStepStepping IMPLEMENTS CNM_CycleManagerInterfaces.ISteppingConfiguration
VAR
	parameters :ICycleManagerStepParameters;
END_VAR

(*

## Short summary
Gets or sets the cycle manager step parameters interface used for stepping configuration.

### Purpose and usage
This property provides access to the underlying cycle manager step parameters interface
that this stepping configurator operates on. It allows getting the current cycle manager instance
and setting a new one if needed for step-specific stepping configuration.

The property is primarily used internally but can be accessed for direct parameter manipulation
or when switching between different cycle manager instances at the step level.

### typical usage patterns
1. **Internal initialization**: Set during configurator setup
2. **Runtime switching**: Change cycle manager instances
3. **Direct access**: Get parameters for advanced step configuration
4. **Dependency injection**: Inject different implementations

### When to use
- During initialization to connect to a cycle manager
- When switching between different cycle manager implementations
- For direct access to step-specific stepping parameters
- In advanced configuration scenarios for individual steps

### Example
```
// Get current cycle manager
VAR
    currentManager : ICycleManagerStepParameters;
END_VAR

currentManager := stepSteppingConfig.cycleManager;

// Check current step stepping state
IF currentManager.currentSteppingEnabled THEN
    // Stepping is enabled for current step
END_IF;

// Set new cycle manager
VAR
    newManager : MyCycleManagerStepImplementation;
END_VAR

stepSteppingConfig.cycleManager := newManager;
```

.. <legal notes>

legal notes
=================
| SPDX-FileCopyrightText: © 2025 ekvip automation GmbH <info@ekvip.de>
| SPDX-License-Identifier: Apache-2.0
| For details check: Apache-2.0_

.. _Apache-2.0: https://www.apache.org/licenses/LICENSE-2.0

.. </legal notes>

*)
PROPERTY cycleManager : ICycleManagerStepParameters
GET
cycleManager := THIS^.parameters;
END_GET
SET
THIS^.parameters := cycleManager;
END_SET
END_PROPERTY

(*

## Short summary
Disables stepping mode for the current cycle manager step.

### Purpose and usage
This method disables the stepping mode functionality for the current step only, overriding
the sequence default. When stepping is disabled for a step, it runs continuously without
requiring manual step triggers, even if the sequence has stepping enabled.

Disabling stepping at the step level is useful for:
- Automated calculations or operations within a stepped sequence
- Time-critical steps that should not wait for triggers
- Background operations that run automatically
- Steps that should always complete without manual intervention

### typical usage patterns
1. **Auto steps**: Steps that run automatically in stepped sequences
2. **Calculations**: Automated computation steps
3. **Fast operations**: Quick steps that don't need manual control
4. **Override sequence**: Disable stepping for specific steps only

### When to use
- For automated steps within a manually stepped sequence
- When specific steps should run without manual triggers
- For calculation or processing steps
- To skip stepping on non-interactive steps

### Example
```
// Disable stepping for calculation step
CASE cycleManager.steps.current OF
    MySteps.MANUAL_SETUP:
        // This step uses sequence stepping settings
        IF setupComplete THEN
            cycleManager.steps.next := MySteps.AUTO_CALCULATION;
        END_IF;
        
    MySteps.AUTO_CALCULATION:
        // Disable stepping for this automated step
        cycleManager.configuration.configuration.step
            .stepping.disable();
        performCalculations();
        IF calculationsComplete THEN
            // Re-enable stepping for next manual step
            cycleManager.configuration.configuration.step
                .stepping.enable();
            cycleManager.steps.next := MySteps.VERIFY_RESULTS;
        END_IF;
END_CASE

// Skip stepping for fast operations
IF isQuickOperation(currentStep) THEN
    cycleManager.configuration.configuration.step
        .stepping.disable();
END_IF;
```

.. <legal notes>

legal notes
=================
| SPDX-FileCopyrightText: © 2025 ekvip automation GmbH <info@ekvip.de>
| SPDX-License-Identifier: Apache-2.0
| For details check: Apache-2.0_

.. _Apache-2.0: https://www.apache.org/licenses/LICENSE-2.0

.. </legal notes>

*)
METHOD disable
THIS^.cycleManager.currentSteppingEnabled := FALSE;
END_METHOD

(*

## Short summary
Enables stepping mode for the current cycle manager step.

### Purpose and usage
This method enables the stepping mode functionality for the current step only, overriding
the sequence default if necessary. When stepping is enabled for a step, execution pauses
after entering the step, requiring manual trigger or auto-step delay before proceeding.

Enabling stepping at the step level is useful for:
- Critical steps requiring verification in automated sequences
- Decision points where operator input is needed
- Steps where results should be inspected
- Debugging specific steps in production sequences

### typical usage patterns
1. **Verification steps**: Force stepping for result checking
2. **Decision points**: Require manual confirmation
3. **Critical operations**: Enable stepping for careful execution
4. **Override sequence**: Enable stepping for specific steps only

### When to use
- For steps requiring operator verification or decision
- During critical operations needing manual control
- At inspection or quality check points
- When specific steps should use stepping regardless of sequence settings

### Example
```
// Enable stepping for verification step
CASE cycleManager.steps.current OF
    MySteps.PERFORM_OPERATION:
        // Normal automated execution
        IF operationComplete THEN
            cycleManager.steps.next := MySteps.VERIFY_RESULTS;
        END_IF;
        
    MySteps.VERIFY_RESULTS:
        // Force stepping for manual verification
        cycleManager.configuration.configuration.step
            .stepping.enable();
        displayResults();
        // Operator must trigger next step manually
        IF resultsApproved THEN
            cycleManager.steps.next := MySteps.CONTINUE;
        END_IF;
END_CASE

// Conditionally enable stepping
IF criticalOperation OR requiresInspection THEN
    cycleManager.configuration.configuration.step
        .stepping.enable();
END_IF;

// Force stepping in production for specific steps
IF isQualityCheckStep(currentStep) AND productionMode THEN
    cycleManager.configuration.configuration.step
        .stepping.enable();  // Override sequence default
END_IF;
```

.. <legal notes>

legal notes
=================
| SPDX-FileCopyrightText: © 2025 ekvip automation GmbH <info@ekvip.de>
| SPDX-License-Identifier: Apache-2.0
| For details check: Apache-2.0_

.. _Apache-2.0: https://www.apache.org/licenses/LICENSE-2.0

.. </legal notes>


*)
METHOD enable
THIS^.cycleManager.currentSteppingEnabled := TRUE;
END_METHOD

END_FUNCTION_BLOCK

// ---- Configurators/classes/CycleManagerDefaultConfigurator.TcPOU
(*

## Short summary
A class to provide fluent access to the default sequence configuration of a cycle manager.

.. <legal notes>

legal notes
=================
| SPDX-FileCopyrightText: © 2024 ekvip automation GmbH <info@ekvip.de>
| SPDX-License-Identifier: Apache-2.0
| For details check: Apache-2.0_

.. _Apache-2.0: https://www.apache.org/licenses/LICENSE-2.0

.. </legal notes>



*)
FUNCTION_BLOCK INTERNAL CycleManagerDefaultConfigurator IMPLEMENTS CNM_CycleManagerInterfaces.ISequenceConfiguration, CNM_CycleManagerInterfaces.IStopRequestConfiguration
VAR
	parameters :CNM_CycleManagerInterfaces.ICycleManagerDefaultParameters;
	steperator :CycleManagerDefaultStepping(); 
	pauserator :CycleManagerDefaultPausing(); 
END_VAR

(*

## Short summary
Sets the stop request behavior to execute after successful step completion.

### Purpose and usage
This method configures the cycle manager to process stop requests only after a step has completed successfully.
When this mode is active, stop requests received during step execution will be deferred until the current step
completes with success.

This ensures that critical operations can complete successfully before the cycle is stopped,
maintaining data integrity and process consistency.

### typical usage patterns
1. **Safe stopping**: Ensure processes complete before stopping
2. **Data consistency**: Finish transactions before stopping
3. **Clean shutdown**: Complete current operation cleanly
4. **Production safety**: Avoid partial operations

### When to use
- When steps must complete successfully before stopping
- For operations that should not be interrupted mid-execution
- When data consistency requires complete transactions
- In production environments requiring clean shutdowns

### Example
```
// Configure safe stopping after success
cycleManager.configuration.configuration.sequence
    .stopRequest
    .afterSuccess();

// Usage in step implementation
CASE cycleManager.steps.current OF
    MySteps.CRITICAL_OPERATION:
        // This operation will complete before stop is processed
        IF performCriticalOperation() THEN
            cycleManager.steps.next := MySteps.NEXT_STEP;
        END_IF;
        // Stop request will be processed after this step succeeds
END_CASE
```

.. <legal notes>

legal notes
=================
| SPDX-FileCopyrightText: © 2025 ekvip automation GmbH <info@ekvip.de>
| SPDX-License-Identifier: Apache-2.0
| For details check: Apache-2.0_

.. _Apache-2.0: https://www.apache.org/licenses/LICENSE-2.0

.. </legal notes>

*)
METHOD afterSuccessfulStep
THIS^.cycleManager.defaultStopRequestMode := CNM_CycleManagerInterfaces.StepStopRequestMode.AFTER_SUCCESSFUL_STEP;
END_METHOD

(*

## Short summary
Gets or sets the cycle manager default parameters interface used by this configurator.

### Purpose and usage
This property provides access to the underlying cycle manager default parameters interface.
It allows getting the current cycle manager instance and setting a new one if needed.

When setting a new cycle manager, all internal configurators (stepping and pausing)
are automatically updated to use the new instance.

### typical usage patterns
1. **Initialization**: Set during configurator creation
2. **Runtime changes**: Switch cycle manager instances
3. **Access parameters**: Get current cycle manager for direct access
4. **Dependency injection**: Inject different implementations

### When to use
- During initialization to set the cycle manager
- When switching between different cycle manager implementations
- For direct access to cycle manager parameters
- In factory patterns for dynamic configuration

### Example
```
// Get current cycle manager
VAR
    currentManager : ICycleManagerDefaultParameters;
END_VAR

currentManager := configurator.cycleManager;

// Set new cycle manager
VAR
    newManager : MyCycleManagerImplementation;
END_VAR

configurator.cycleManager := newManager;
// All sub-configurators now use newManager

// Direct parameter access
IF configurator.cycleManager.defaultTimeout > T#10S THEN
    // Handle long timeout
END_IF;
```

.. <legal notes>

legal notes
=================
| SPDX-FileCopyrightText: © 2025 ekvip automation GmbH <info@ekvip.de>
| SPDX-License-Identifier: Apache-2.0
| For details check: Apache-2.0_

.. _Apache-2.0: https://www.apache.org/licenses/LICENSE-2.0

.. </legal notes>


*)
PROPERTY cycleManager : CNM_CycleManagerInterfaces.ICycleManagerDefaultParameters
GET
cycleManager := THIS^.parameters;
END_GET
SET
THIS^.parameters := cycleManager;
THIS^.steperator.cycleManager := THIS^.cycleManager;
THIS^.pauserator.cycleManager := THIS^.cycleManager;
END_SET
END_PROPERTY

(*

## Short summary
This property sets the next step in case of an error.
Is reset to the default ERROR_STEP when the current step changes.

.. <legal notes>

legal notes
=================
| SPDX-FileCopyrightText: © 2024 ekvip automation GmbH <info@ekvip.de>
| SPDX-License-Identifier: Apache-2.0
| For details check: Apache-2.0_

.. _Apache-2.0: https://www.apache.org/licenses/LICENSE-2.0

.. </legal notes>

*)
PROPERTY errorStep : DINT
SET
THIS^.cycleManager.defaultErrorStep := errorStep;
END_SET
END_PROPERTY

(*

## Short summary
Initializes the CycleManagerDefaultConfigurator and its sub-configurators.

.. <legal notes>

legal notes
=================
| SPDX-FileCopyrightText: © 2025 ekvip automation GmbH <info@ekvip.de>
| SPDX-License-Identifier: Apache-2.0
| For details check: Apache-2.0_

.. _Apache-2.0: https://www.apache.org/licenses/LICENSE-2.0

.. </legal notes>

*)
//FB_Init is always available implicitly and it is used primarily for initialization.
//The return value is not evaluated. For a specific influence, you can also declare the
//methods explicitly and provide additional code there with the standard initialization
//code. You can evaluate the return value.
METHOD FB_Init: BOOL
VAR_INPUT
    bInitRetains: BOOL; // TRUE: the retain variables are initialized (reset warm / reset cold)
    bInCopyCode: BOOL;  // TRUE: the instance will be copied to the copy code afterward (online change)   
END_VAR
THIS^.steperator.cycleManager := THIS^.cycleManager;
THIS^.pauserator.cycleManager := THIS^.cycleManager;
END_METHOD

(*

## Short summary
Sets the stop request behavior to ignore all stop requests.

### Purpose and usage
This method configures the cycle manager to completely ignore all stop requests.
When this mode is active, stop requests will not be processed at all, and the cycle
will continue running until completion or until an error occurs.

This mode should be used with caution as it prevents normal stopping mechanisms
from working.

### typical usage patterns
1. **Critical sequences**: Operations that must not be interrupted
2. **Atomic operations**: Multi-step processes that must complete
3. **Safety sequences**: Emergency procedures that must finish
4. **Calibration routines**: Procedures that cannot be stopped

### When to use
- For critical operations that must complete without interruption
- During safety-critical sequences
- For atomic multi-step operations
- When implementing non-interruptible calibration routines
- Use with extreme caution - limits operator control

### Example
```
// Configure to ignore stop requests
cycleManager.configuration.configuration.sequence
    .stopRequest
    .ignore();

// Usage in critical sequence
CASE cycleManager.steps.current OF
    MySteps.CRITICAL_SEQUENCE_START:
        // Configure to ignore stops for critical sequence
        cycleManager.configuration.configuration.sequence
            .stopRequest.ignore();
        cycleManager.steps.next := MySteps.CRITICAL_STEP_1;
        
    MySteps.CRITICAL_SEQUENCE_END:
        // Re-enable stop handling after critical sequence
        cycleManager.configuration.configuration.sequence
            .stopRequest.afterSuccess();
        cycleManager.steps.next := MySteps.NORMAL_OPERATION;
END_CASE

// Stop requests during critical sequence will be ignored
IF stopButton THEN
    cycleManager.requestStop();  // Has no effect when ignore is active
END_IF;
```

.. <legal notes>

legal notes
=================
| SPDX-FileCopyrightText: © 2025 ekvip automation GmbH <info@ekvip.de>
| SPDX-License-Identifier: Apache-2.0
| For details check: Apache-2.0_

.. _Apache-2.0: https://www.apache.org/licenses/LICENSE-2.0

.. </legal notes>

*)
METHOD ignore
THIS^.cycleManager.defaultStopRequestMode := CNM_CycleManagerInterfaces.StepStopRequestMode.IGNORE;
END_METHOD

(*

## Short summary
Sets the stop request behavior to always process stop requests immediately.

### Purpose and usage
This method configures the cycle manager to always process stop requests immediately,
regardless of the current step's execution state or outcome. Stop requests are handled
as soon as they are received, potentially interrupting the current operation.

This mode provides the most responsive stop behavior but may interrupt operations
that are in progress.

### typical usage patterns
1. **Emergency stops**: Immediate response to stop requests
2. **Non-critical operations**: When interruption is acceptable
3. **Debug mode**: Quick stopping during development
4. **User-initiated stops**: Responsive UI behavior

### When to use
- When immediate stop response is critical
- For non-critical operations that can be interrupted
- During development and debugging
- When user experience requires immediate feedback
- In emergency stop scenarios

### Example
```
// Configure immediate stop processing
cycleManager.configuration.configuration.sequence
    .stopRequest
    .always();

// Usage with emergency stop
IF emergencyStopButton THEN
    cycleManager.requestStop();  // Will be processed immediately
END_IF;

// In step implementation
CASE cycleManager.steps.current OF
    MySteps.LONG_OPERATION:
        // This operation can be interrupted at any time
        performLongOperation();
        // Stop request processed immediately if received
END_CASE
```

.. <legal notes>

legal notes
=================
| SPDX-FileCopyrightText: © 2025 ekvip automation GmbH <info@ekvip.de>
| SPDX-License-Identifier: Apache-2.0
| For details check: Apache-2.0_

.. _Apache-2.0: https://www.apache.org/licenses/LICENSE-2.0

.. </legal notes>

*)
METHOD immediate
THIS^.cycleManager.defaultStopRequestMode := CNM_CycleManagerInterfaces.StepStopRequestMode.IMMEDIATE;
END_METHOD

(*

## Short summary
This method sets the stop request behaviour to ``StepStopRequestMode.AFTER_NOT_SUCCESS``.

.. <legal notes>

legal notes
=================
| SPDX-FileCopyrightText: © 2024 ekvip automation GmbH <info@ekvip.de>
| SPDX-License-Identifier: Apache-2.0
| For details check: Apache-2.0_

.. _Apache-2.0: https://www.apache.org/licenses/LICENSE-2.0

.. </legal notes>

*)
METHOD onBusy
THIS^.cycleManager.defaultStopRequestMode := CNM_CycleManagerInterfaces.StepStopRequestMode.ON_BUSY;
END_METHOD

(*

## Short summary
Provides access to the pause configuration for the cycle manager sequence.

### Purpose and usage
This property returns the pause configuration interface that allows setting pause-related
parameters for the entire sequence. It provides a fluent interface for configuring how
the cycle manager handles pause requests.

The pause configuration controls:
- Whether pausing is allowed
- Pause timeout behavior
- Resume conditions
- Pause state handling


### typical usage patterns
1. **Enable/disable pausing**: Control if sequence can be paused
2. **Set pause timeouts**: Define maximum pause duration
3. **Configure resume**: Set conditions for resuming
4. **Pause behavior**: Define what happens during pause

### When to use
- To enable or disable pause functionality
- When setting pause timeout limits
- For configuring pause/resume behavior
- To implement operator-controlled pausing

### Example
```
// Enable pausing with timeout
cycleManager.configuration.configuration.sequence
    .pause
    .enabled(TRUE)
    .timeout(T#30S);

// Disable pausing for critical operations
cycleManager.configuration.configuration.sequence
    .pause
    .enabled(FALSE);

// Configure pause with auto-resume
cycleManager.configuration.configuration.sequence
    .pause
    .enabled(TRUE)
    .autoResume(TRUE)
    .autoResumeDelay(T#5S);
```

.. <legal notes>

legal notes
=================
| SPDX-FileCopyrightText: © 2025 ekvip automation GmbH <info@ekvip.de>
| SPDX-License-Identifier: Apache-2.0
| For details check: Apache-2.0_

.. _Apache-2.0: https://www.apache.org/licenses/LICENSE-2.0

.. </legal notes>

*)
PROPERTY pause : CNM_CycleManagerInterfaces.IPauseConfiguration
GET
pause := pauserator;
END_GET
END_PROPERTY

(*

## Short summary
Specifies whether the SUCCESS step of the state machine can be skipped when the transition condition to SUCCESS is already fulfilled.

When set to false, the state machine immediately returns SUCCESS as soon as the transition condition to the SUCCESS state is met, 
without executing the dedicated SUCCESS step. This optimization can save one execution cycle per state machine invocation, which is 
especially beneficial in nested or complex state machine structures.

When set to true, the SUCCESS step will always be executed at least once before the state machine returns SUCCESS. This is required 
in cases where the SUCCESS step performs essential actions (e.g., resetting outputs, logging, or cleanup).

The default value is false.

### Use Case
Use false when the SUCCESS step has no functional side effects and skipping it can improve performance.
Use true when the SUCCESS step contains logic that must be executed explicitly.

.. <legal notes>

legal notes
=================
| SPDX-FileCopyrightText: © 2025 ekvip automation GmbH <info@ekvip.de>
| SPDX-License-Identifier: Apache-2.0
| For details check: Apache-2.0_

.. _Apache-2.0: https://www.apache.org/licenses/LICENSE-2.0

.. </legal notes>

*)

PROPERTY requireSuccessStep : BOOL
SET
THIS^.parameters.defaultRequireSuccessStep := requireSuccessStep;
END_SET
END_PROPERTY

(*

## Short summary
Provides access to the stepping configuration for the cycle manager sequence.

### Purpose and usage
This property returns the stepping configuration interface that allows setting stepping-related
parameters for the entire sequence. It provides a fluent interface for configuring step-by-step
execution mode, typically used for debugging and commissioning.

The stepping configuration controls:
- Whether stepping mode is enabled
- Auto-step delays
- Step trigger conditions
- Single-step behavior


### typical usage patterns
1. **Debug mode**: Enable step-by-step execution
2. **Commissioning**: Test sequences one step at a time
3. **Auto-stepping**: Configure automatic step advancement
4. **Manual control**: Require operator confirmation per step

### When to use
- During commissioning and debugging
- For training operators on sequence flow
- When testing new sequences step-by-step
- For troubleshooting sequence issues

### Example
```
// Enable manual stepping mode
cycleManager.configuration.configuration.sequence
    .stepping
    .enabled(TRUE)
    .autoStep(FALSE);

// Enable auto-stepping with delay
cycleManager.configuration.configuration.sequence
    .stepping
    .enabled(TRUE)
    .autoStep(TRUE)
    .autoStepDelay(T#2S);

// Disable stepping for production
cycleManager.configuration.configuration.sequence
    .stepping
    .enabled(FALSE);

// Conditional stepping based on mode
IF commissioningMode THEN
    cycleManager.configuration.configuration.sequence
        .stepping.enabled(TRUE);
END_IF;
```

.. <legal notes>

legal notes
=================
| SPDX-FileCopyrightText: © 2025 ekvip automation GmbH <info@ekvip.de>
| SPDX-License-Identifier: Apache-2.0
| For details check: Apache-2.0_

.. _Apache-2.0: https://www.apache.org/licenses/LICENSE-2.0

.. </legal notes>

*)
PROPERTY stepping : CNM_CycleManagerInterfaces.ISteppingConfiguration
GET
VAR_INST
END_VAR
stepping := steperator;
END_GET
END_PROPERTY

(*

## Short summary
Sets the default step width for automatic step increments in the sequence.

### Purpose and usage
This property sets the default increment value used when automatically advancing to the next step.
When no explicit next step is specified, the cycle manager will advance by this step width value.

Typical step widths:
- 1: Sequential step execution (most common)
- 10: Grouped steps with room for insertions
- 100: Major phase transitions
- Custom values for specific sequencing needs

### typical usage patterns
1. **Sequential execution**: Set to 1 for normal flow
2. **Grouped steps**: Use larger values for step groups
3. **Phase transitions**: Large values between phases
4. **Custom sequences**: Application-specific increments

### When to use
- When implementing non-sequential step numbering
- For organizing steps into logical groups
- To leave room for future step insertions
- When matching legacy step numbering systems

### Example
```
// Standard sequential execution
cycleManager.configuration.configuration.sequence
    .stepWidth := 1;

// Grouped steps with room for expansion
cycleManager.configuration.configuration.sequence
    .stepWidth := 10;
    
// Step implementation
CASE cycleManager.steps.current OF
    100:  // Phase 1 start
        doPhase1Init();
        // Automatically advances to 110
        
    110:  // Phase 1 operation
        doPhase1Operation();
        // Automatically advances to 120
        
    200:  // Phase 2 start (explicit jump needed)
        doPhase2Init();
        // Automatically advances to 210
END_CASE
``` 

.. <legal notes>

legal notes
=================
| SPDX-FileCopyrightText: © 2025 ekvip automation GmbH <info@ekvip.de>
| SPDX-License-Identifier: Apache-2.0
| For details check: Apache-2.0_

.. _Apache-2.0: https://www.apache.org/licenses/LICENSE-2.0

.. </legal notes>


*)
PROPERTY stepWidth : DINT
SET
THIS^.cycleManager.defaultStepWidth := stepWidth;
END_SET
END_PROPERTY

(*

## Short summary
Provides access to the stop request configuration interface.

### Purpose and usage
This property returns the stop request configuration interface, providing access to methods
that configure how the cycle manager handles stop requests. The configurator itself implements
the IStopRequestConfiguration interface.

Available configuration modes:
- always(): Process stop requests immediately
- afterSuccess(): Process after successful step completion
- afterNotSuccess(): Process after unsuccessful step completion
- ignore(): Ignore all stop requests


### typical usage patterns
1. **Fluent configuration**: Chain stop configuration methods
2. **Mode selection**: Choose appropriate stop handling
3. **Dynamic configuration**: Change modes during runtime
4. **Safety configuration**: Set safe stop behavior

### When to use
- To configure stop request handling behavior
- When implementing different stop strategies
- For safety-critical stop configurations
- During mode-dependent stop handling

### Example
```
// Configure stop after success
cycleManager.configuration.configuration.sequence
    .stopRequest
    .afterSuccess();

// Configure immediate stop
cycleManager.configuration.configuration.sequence
    .stopRequest
    .always();

// Chain with other configurations
cycleManager.configuration.configuration.sequence
    .timeout := T#10S;
    .stopRequest.afterSuccess();
    .pause.enabled(TRUE);

// Dynamic configuration based on mode
IF emergencyMode THEN
    cycleManager.configuration.configuration.sequence
        .stopRequest.always();
ELSE
    cycleManager.configuration.configuration.sequence
        .stopRequest.afterSuccess();
END_IF;
```

.. <legal notes>

legal notes
=================
| SPDX-FileCopyrightText: © 2025 ekvip automation GmbH <info@ekvip.de>
| SPDX-License-Identifier: Apache-2.0
| For details check: Apache-2.0_

.. _Apache-2.0: https://www.apache.org/licenses/LICENSE-2.0

.. </legal notes>

*)
PROPERTY stopRequest : CNM_CycleManagerInterfaces.IStopRequestConfiguration
GET
stopRequest := THIS^;
END_GET
END_PROPERTY

(*

## Short summary
This property sets the maximum execution time for the current step. 
The cycle manager will go into the error step after the time elapsed.
Set to T#0MS for no timeout.

.. <legal notes>

legal notes
=================
| SPDX-FileCopyrightText: © 2024 ekvip automation GmbH <info@ekvip.de>
| SPDX-License-Identifier: Apache-2.0
| For details check: Apache-2.0_

.. _Apache-2.0: https://www.apache.org/licenses/LICENSE-2.0

.. </legal notes>

*)
PROPERTY timeout : TIME
SET
THIS^.cycleManager.defaultTimeout := timeout;
END_SET
END_PROPERTY

(*

## Short summary
This property sets the step that will be set if the current step reaches a timeout. 
Will by default be the error step and reset after the current step changes.

.. <legal notes>

legal notes
=================
| SPDX-FileCopyrightText: © 2024 ekvip automation GmbH <info@ekvip.de>
| SPDX-License-Identifier: Apache-2.0
| For details check: Apache-2.0_

.. _Apache-2.0: https://www.apache.org/licenses/LICENSE-2.0

.. </legal notes>

*)
PROPERTY timeoutStep : DINT
SET
THIS^.cycleManager.defaultTimeoutStep := timeoutStep;
END_SET
END_PROPERTY

END_FUNCTION_BLOCK

// ---- Configurators/classes/CycleManagerDefaultStepping.TcPOU
(*

## Short summary
A class to provide fluent access to the default stepping sequence configuration of a cycle manager.

.. <legal notes>

legal notes
=================
| SPDX-FileCopyrightText: © 2024 ekvip automation GmbH <info@ekvip.de>
| SPDX-License-Identifier: Apache-2.0
| For details check: Apache-2.0_

.. _Apache-2.0: https://www.apache.org/licenses/LICENSE-2.0

.. </legal notes>



*)
FUNCTION_BLOCK INTERNAL CycleManagerDefaultStepping IMPLEMENTS CNM_CycleManagerInterfaces.ISteppingConfiguration
VAR
	parameters :CNM_CycleManagerInterfaces.ICycleManagerDefaultParameters;
END_VAR

(*

## Short summary
Gets or sets the cycle manager default parameters interface used for stepping configuration.

### Purpose and usage
This property provides access to the underlying cycle manager default parameters interface
that this stepping configurator operates on. It allows getting the current cycle manager instance
and setting a new one if needed.

The property is primarily used internally but can be accessed for direct parameter manipulation
or when switching between different cycle manager instances.

### typical usage patterns
1. **Internal initialization**: Set during configurator setup
2. **Runtime switching**: Change cycle manager instances
3. **Direct access**: Get parameters for advanced configuration
4. **Dependency injection**: Inject different implementations

### When to use
- During initialization to connect to a cycle manager
- When switching between different cycle manager implementations
- For direct access to stepping-related parameters
- In advanced configuration scenarios

### Example
```
// Get current cycle manager
VAR
    currentManager : ICycleManagerDefaultParameters;
END_VAR

currentManager := steppingConfig.cycleManager;

// Check current stepping state
IF currentManager.defaultSteppingEnabled THEN
    // Stepping is enabled
END_IF;

// Set new cycle manager
VAR
    newManager : MyCycleManagerImplementation;
END_VAR

steppingConfig.cycleManager := newManager;
```

.. <legal notes>

legal notes
=================
| SPDX-FileCopyrightText: © 2025 ekvip automation GmbH <info@ekvip.de>
| SPDX-License-Identifier: Apache-2.0
| For details check: Apache-2.0_

.. _Apache-2.0: https://www.apache.org/licenses/LICENSE-2.0

.. </legal notes>

*)
PROPERTY cycleManager : CNM_CycleManagerInterfaces.ICycleManagerDefaultParameters
GET
cycleManager := THIS^.parameters;
END_GET
SET
THIS^.parameters := cycleManager;
END_SET
END_PROPERTY

(*

## Short summary
Disables stepping mode for the cycle manager sequence.

### Purpose and usage
This method disables the stepping mode functionality for the entire cycle manager sequence.
When stepping is disabled, the cycle runs continuously without requiring manual step triggers,
executing each step automatically as conditions are met.

Disabling stepping mode is the normal production configuration where sequences run
automatically from start to finish.

### typical usage patterns
1. **Production mode**: Disable stepping for automatic execution
2. **Normal operation**: Run sequences without manual intervention
3. **Automated testing**: Execute full sequences automatically
4. **Performance mode**: Remove stepping overhead

### When to use
- In production environments for automatic operation
- When commissioning is complete and manual control not needed
- For automated test sequences
- When maximum performance is required
- As the default mode for normal operation

### Example
```
// Disable stepping for production
cycleManager.configuration.configuration.sequence
    .stepping
    .disable();

// Switch modes based on operation
IF productionMode THEN
    cycleManager.configuration.configuration.sequence
        .stepping.disable();
ELSE
    cycleManager.configuration.configuration.sequence
        .stepping.enable();
END_IF;

// Ensure stepping is disabled for critical sequences
CASE cycleManager.steps.current OF
    MySteps.CRITICAL_SEQUENCE_START:
        cycleManager.configuration.configuration.sequence
            .stepping.disable();  // No manual stepping allowed
        cycleManager.steps.next := MySteps.CRITICAL_OPERATION;
END_CASE

// Update HMI based on stepping mode
IF NOT cycleManager.steppingEnabled THEN
    HMI.StepButton.Visible := FALSE;
    HMI.AutoStepCheckbox.Visible := FALSE;
END_IF;
```

.. <legal notes>

legal notes
=================
| SPDX-FileCopyrightText: © 2025 ekvip automation GmbH <info@ekvip.de>
| SPDX-License-Identifier: Apache-2.0
| For details check: Apache-2.0_

.. _Apache-2.0: https://www.apache.org/licenses/LICENSE-2.0

.. </legal notes>

*)
METHOD disable
THIS^.cycleManager.defaultSteppingEnabled := FALSE;
END_METHOD

(*

## Short summary
Enables stepping mode for the cycle manager sequence.

### Purpose and usage
This method enables the stepping mode functionality for the entire cycle manager sequence.
When stepping is enabled, the cycle execution pauses after each step, requiring manual
trigger or auto-step delay before proceeding to the next step.

Stepping mode is essential for:
- Commissioning new sequences
- Debugging sequence logic
- Training operators
- Validating step transitions

### typical usage patterns
1. **Commissioning**: Step through new sequences manually
2. **Debugging**: Examine state between steps
3. **Training**: Demonstrate sequence flow to operators
4. **Validation**: Verify each step executes correctly

### When to use
- During initial commissioning of new equipment
- When debugging sequence problems
- For operator training sessions
- During sequence development and testing
- When validating modifications to sequences

### Example
```
// Enable stepping for commissioning
cycleManager.configuration.configuration.sequence
    .stepping
    .enable();

// Enable stepping with auto-advance
IF debugMode THEN
    cycleManager.configuration.configuration.sequence
        .stepping.enable();
    cycleManager.setAutoStepDelay(T#2S);  // Auto advance every 2 seconds
END_IF;

// Manual step control
IF cycleManager.steppingEnabled THEN
    IF HMI.StepButton.Pressed THEN
        cycleManager.triggerStep();  // Advance to next step
    END_IF;
END_IF;

// Show stepping controls in HMI
IF cycleManager.steppingEnabled THEN
    HMI.StepButton.Visible := TRUE;
    HMI.CurrentStep.Text := INT_TO_STRING(cycleManager.steps.current);
    HMI.NextStep.Text := INT_TO_STRING(cycleManager.steps.next);
END_IF;
```

.. <legal notes>

legal notes
=================
| SPDX-FileCopyrightText: © 2025 ekvip automation GmbH <info@ekvip.de>
| SPDX-License-Identifier: Apache-2.0
| For details check: Apache-2.0_

.. _Apache-2.0: https://www.apache.org/licenses/LICENSE-2.0

.. </legal notes>

*)
METHOD enable
THIS^.cycleManager.defaultSteppingEnabled := TRUE;
END_METHOD

END_FUNCTION_BLOCK

// ---- Configurators/classes/CycleManagerDefaultPausing.TcPOU
(*

## Short summary
A class to provide fluent access to the default sequence pausing configuration of a cycle manager.

.. <legal notes>

legal notes
=================
| SPDX-FileCopyrightText: © 2024 ekvip automation GmbH <info@ekvip.de>
| SPDX-License-Identifier: Apache-2.0
| For details check: Apache-2.0_

.. _Apache-2.0: https://www.apache.org/licenses/LICENSE-2.0

.. </legal notes>



*)
FUNCTION_BLOCK INTERNAL CycleManagerDefaultPausing IMPLEMENTS CNM_CycleManagerInterfaces.IPauseConfiguration
VAR
	parameters :CNM_CycleManagerInterfaces.ICycleManagerDefaultParameters;
END_VAR

(*

## Short summary
Gets or sets the cycle manager default parameters interface used for pause configuration.

### Purpose and usage
This property provides access to the underlying cycle manager default parameters interface
that this pause configurator operates on. It allows getting the current cycle manager instance
and setting a new one if needed.

The property is primarily used internally but can be accessed for direct parameter manipulation
or when switching between different cycle manager instances.

### typical usage patterns
1. **Internal initialization**: Set during configurator setup
2. **Runtime switching**: Change cycle manager instances
3. **Direct access**: Get parameters for advanced configuration
4. **Dependency injection**: Inject different implementations

### When to use
- During initialization to connect to a cycle manager
- When switching between different cycle manager implementations
- For direct access to pause-related parameters
- In advanced configuration scenarios

### Example
```
// Get current cycle manager
VAR
    currentManager : ICycleManagerDefaultParameters;
END_VAR

currentManager := pauseConfig.cycleManager;

// Check current pause state
IF currentManager.defaultPauseEnabled THEN
    // Pause is enabled
END_IF;

// Set new cycle manager
VAR
    newManager : MyCycleManagerImplementation;
END_VAR

pauseConfig.cycleManager := newManager;
```

.. <legal notes>

legal notes
=================
| SPDX-FileCopyrightText: © 2025 ekvip automation GmbH <info@ekvip.de>
| SPDX-License-Identifier: Apache-2.0
| For details check: Apache-2.0_

.. _Apache-2.0: https://www.apache.org/licenses/LICENSE-2.0

.. </legal notes>

*)
PROPERTY cycleManager : CNM_CycleManagerInterfaces.ICycleManagerDefaultParameters
GET
cycleManager := THIS^.parameters;
END_GET
SET
THIS^.parameters := cycleManager;
END_SET
END_PROPERTY

(*

## Short summary
Disables pause functionality for the cycle manager sequence.

### Purpose and usage
This method disables the pause functionality for the entire cycle manager sequence.
When pause is disabled, pause requests will be ignored and the cycle will continue
running without interruption.

Disabling pause is useful for:
- Critical operations that must not be interrupted
- Production mode where pausing is not desired
- Automated sequences that should run to completion
- Safety-critical procedures

### typical usage patterns
1. **Production mode**: Disable pause in normal operation
2. **Critical sequences**: Prevent interruption of important operations
3. **Automated runs**: Ensure uninterrupted execution
4. **Safety procedures**: Prevent unsafe pausing

### When to use
- In production environments where pausing should not be allowed
- During critical operations that must complete
- For automated sequences that should not be interrupted
- When implementing safety-critical procedures

### Example
```
// Disable pause for production
cycleManager.configuration.configuration.sequence
    .pause
    .disable();

// Temporarily disable pause for critical operation
CASE cycleManager.steps.current OF
    MySteps.CRITICAL_START:
        cycleManager.configuration.configuration.sequence
            .pause.disable();
        cycleManager.steps.next := MySteps.CRITICAL_OPERATION;
        
    MySteps.CRITICAL_END:
        cycleManager.configuration.configuration.sequence
            .pause.enable();  // Re-enable after critical section
        cycleManager.steps.next := MySteps.NORMAL_OPERATION;
END_CASE

// Check if pause is disabled
IF NOT cycleManager.pauseEnabled THEN
    HMI.PauseButton.Enabled := FALSE;
END_IF;
```

.. <legal notes>

legal notes
=================
| SPDX-FileCopyrightText: © 2025 ekvip automation GmbH <info@ekvip.de>
| SPDX-License-Identifier: Apache-2.0
| For details check: Apache-2.0_

.. _Apache-2.0: https://www.apache.org/licenses/LICENSE-2.0

.. </legal notes>

*)
METHOD disable
THIS^.cycleManager.defaultPauseEnabled := FALSE;
END_METHOD

(*

## Short summary
Enables pause functionality for the cycle manager sequence.

### Purpose and usage
This method enables the pause functionality for the entire cycle manager sequence.
When pause is enabled, the cycle can be paused at appropriate points, allowing operators
to temporarily halt execution and resume later.

Enabling pause is useful for:
- Manual control during commissioning
- Debugging and troubleshooting
- Operator-controlled production
- Training and demonstration

### typical usage patterns
1. **Commissioning mode**: Enable pause for manual control
2. **Debug mode**: Allow pausing for troubleshooting
3. **Training**: Enable pause for step-by-step demonstration
4. **Semi-automatic mode**: Operator-controlled execution

### When to use
- During commissioning and testing phases
- In debug or maintenance modes
- For operator training scenarios
- When manual intervention might be needed
- In semi-automatic operation modes

### Example
```
// Enable pause for commissioning
cycleManager.configuration.configuration.sequence
    .pause
    .enable();

// Enable pause based on operation mode
IF commissioningMode OR debugMode THEN
    cycleManager.configuration.configuration.sequence
        .pause.enable();
ELSE
    cycleManager.configuration.configuration.sequence
        .pause.disable();
END_IF;

// Use with HMI controls
IF cycleManager.pauseEnabled THEN
    HMI.PauseButton.Enabled := TRUE;
    HMI.ResumeButton.Enabled := cycleManager.isPaused;
END_IF;

// Handle pause request
IF HMI.PauseButton.Pressed AND cycleManager.pauseEnabled THEN
    cycleManager.requestPause();
END_IF;
```

.. <legal notes>

legal notes
=================
| SPDX-FileCopyrightText: © 2025 ekvip automation GmbH <info@ekvip.de>
| SPDX-License-Identifier: Apache-2.0
| For details check: Apache-2.0_

.. _Apache-2.0: https://www.apache.org/licenses/LICENSE-2.0

.. </legal notes>

*)
METHOD enable
THIS^.cycleManager.defaultPauseEnabled := TRUE;
END_METHOD

END_FUNCTION_BLOCK

// ---- CycleManager/classes/AbstractCycleManager.TcPOU
(*

## Short summary
An abstract CycleManager implementation to provide basic functionality.
Does not update the state of the cyclemanager, it only provides some protected update functions.

.. <info>
If used in the same step, the order/precedence of method calls should be like this:
configurations
enter
executeCommand
evaluate
waitFor
proceed
proceedWith
acknowledge
leave
.. </info>

.. <legal notes>

legal notes
=================
| SPDX-FileCopyrightText: © 2024 ekvip automation GmbH <info@ekvip.de>
| SPDX-License-Identifier: Apache-2.0
| For details check: Apache-2.0_

.. _Apache-2.0: https://www.apache.org/licenses/LICENSE-2.0

.. </legal notes>



*)
FUNCTION_BLOCK ABSTRACT AbstractCycleManager 
EXTENDS CNM_AssertionInterfaces.AbstractAssertor 
IMPLEMENTS CNM_CycleManagerInterfaces.ISingleExecutionCycleManager, 
	CNM_CycleManagerInterfaces.ICycleManagerDefaultParameters, 
	ICycleManagerStepParameters
//config
VAR
	sequenceErrorStep :DINT := STEP_ERROR;
	sequencePauseEnabled :BOOL := FALSE;
	sequenceSteppingEnabled :BOOL := FALSE;
	sequenceTimeOut :TIME := T#0S;
	sequenceStopRequestMode :CNM_CycleManagerInterfaces.StepStopRequestMode := CNM_CycleManagerInterfaces.StepStopRequestMode.IGNORE;
	sequenceTimeoutStep :DINT := STEP_ERROR;
	sequenceStepWidth :DINT := 1;
	sequenceRequireSuccessStep :BOOL := FALSE;
	
	stepErrorStep :DINT := STEP_ERROR;
	stepPauseEnabled :BOOL := FALSE;
	stepSteppingEnabled :BOOL := FALSE;
	stepTimeOut :TIME := T#0S;
	stepCurrentStopRequestMode :CNM_CycleManagerInterfaces.StepStopRequestMode := CNM_CycleManagerInterfaces.StepStopRequestMode.IGNORE;
	stepTimeoutStep :DINT := STEP_ERROR;
	stepStepWidth :DINT := 1;
END_VAR
VAR
	lastStepBeforePause : DINT;
	lastStep : DINT;
	
	currentStep : DINT := CNM_ReturnTypes.DefaultSteps.STEP.IDLE;
	nextStep : DINT := CNM_ReturnTypes.DefaultSteps.STEP.IDLE;
	nextStepSpecifiedByUser :BOOL := FALSE;
	lastExecute : BOOL;
	externalExecute : BOOL;
	currentState : CNM_ReturnTypes.SingleExecutionState := CNM_ReturnTypes.SingleExecutionState.IDLE;
	wasError : BOOL;
	wasTimeoutError : BOOL;
	gotHereByError : BOOL;
	stepLastCycle : DINT;
	wasNotSuccess: BOOL;
	wasSuccess: BOOL;
	firstCycle : BOOL;
	timeoutTimer : TON;
	
	//used for cycle time optimizations
	registeredEnter : BOOL;
	registeredCommand : BOOL;
	registeredEval : BOOL;
	registeredLeave : BOOL;	
END_VAR
VAR CONSTANT
	STEP_IDLE :DINT := CNM_ReturnTypes.DefaultSteps.STEP.IDLE;
	STEP_INIT :DINT := CNM_ReturnTypes.DefaultSteps.STEP.INIT;
	STEP_ERROR :DINT := CNM_ReturnTypes.DefaultSteps.STEP.ERROR;
	STEP_ABORT :DINT := CNM_ReturnTypes.DefaultSteps.STEP.ABORT;
	STEP_PAUSE :DINT := CNM_ReturnTypes.DefaultSteps.STEP.PAUSE;
	STEP_SUCCESS :DINT := CNM_ReturnTypes.DefaultSteps.STEP.SUCCESS;	
END_VAR


(*

## Short summary
This method acknowledges an error in the state machine and resets the current step to the step befor the error occured.

.. <legal notes>

legal notes
=================
| SPDX-FileCopyrightText: © 2024 ekvip automation GmbH <info@ekvip.de>
| SPDX-License-Identifier: Apache-2.0
| For details check: Apache-2.0_

.. _Apache-2.0: https://www.apache.org/licenses/LICENSE-2.0

.. </legal notes>

*)
{attribute 'hide'}
METHOD acknowledge
IF(THIS^.gotHereByError)THEN
	THIS^.next := THIS^.last;
	THIS^.wasNotSuccess := FALSE;
	THIS^.wasError := FALSE;
	THIS^.wasTimeoutError := FALSE;
	THIS^.wasSuccess := TRUE;
END_IF
END_METHOD

(*

## Short summary
This method is called if an assertion was ``FALSE``

.. <legal notes>

legal notes
=================
| SPDX-FileCopyrightText: © 2022 ekvip automation GmbH <info@ekvip.de>
| SPDX-License-Identifier: Apache-2.0
| For details check: Apache-2.0_

.. _Apache-2.0: https://www.apache.org/licenses/LICENSE-2.0

.. </legal notes>


*)
METHOD assertionWasWrong
VAR_INPUT
	(* caller object of the method *)
	caller	: CNM_AbstractObject.IObject;
	(* alarm message *)
	message	: CNM_AssertionInterfaces.AssertMessage;
	(* debugging information *)
	additionalText	: Tc2_System.T_MaxString;
END_VAR
THIS^.wasError := TRUE;
THIS^.wasSuccess := FALSE;
THIS^.wasNotSuccess := TRUE;
END_METHOD

(*

## Short summary
An interface to provide configurations for cycle manager in a fluent way.

.. <legal notes>

legal notes
=================
| SPDX-FileCopyrightText: © 2024 ekvip automation GmbH <info@ekvip.de>
| SPDX-License-Identifier: Apache-2.0
| For details check: Apache-2.0_

.. _Apache-2.0: https://www.apache.org/licenses/LICENSE-2.0

.. </legal notes>



*)
PROPERTY configuration : CNM_CycleManagerInterfaces.ICycleManagerConfigurationScope
GET
VAR_INST
	configurator :CycleManagerConfigurator(THIS^, THIS^);
END_VAR
configuration := configurator;
END_GET
END_PROPERTY

(*

## Short summary
This property returns the current step of the cycle manager.
Proposed use is as CASE control.

### Example
```
CASE cyclemanager.steps.current OF
DefaultSteps.STEP.IDLE:
	;
DefaultSteps.STEP.INIT:
	;
2:
	;
3:
	;
4:
	;
DefaultSteps.STEP.SUCCESS:
	;
DefaultSteps.STEP.ERROR:
	;
DefaultSteps.STEP.ABORT:
	;
ELSE ;
END_CASE
```

.. <legal notes>

legal notes
=================
| SPDX-FileCopyrightText: © 2024 ekvip automation GmbH <info@ekvip.de>
| SPDX-License-Identifier: Apache-2.0
| For details check: Apache-2.0_

.. _Apache-2.0: https://www.apache.org/licenses/LICENSE-2.0

.. </legal notes>

*)
{attribute 'hide'}
PROPERTY current : DINT
GET
current := THIS^.currentStep;
END_GET
SET // PRIVATE
THIS^.currentStep := current;
END_SET
END_PROPERTY

{attribute 'hide'}
PROPERTY currentErrorStep : DINT
GET // PROTECTED
currentErrorStep := THIS^.stepErrorStep;
END_GET
SET
THIS^.stepErrorStep := currentErrorStep;
END_SET
END_PROPERTY

{attribute 'hide'}
PROPERTY currentPauseEnabled : BOOL
GET // PROTECTED
currentPauseEnabled := THIS^.stepPauseEnabled;
END_GET
SET
THIS^.stepPauseEnabled := currentPauseEnabled;
END_SET
END_PROPERTY

{attribute 'hide'}
PROPERTY currentSteppingEnabled : BOOL
GET // PROTECTED
currentSteppingEnabled := THIS^.stepSteppingEnabled;
END_GET
SET
THIS^.stepSteppingEnabled := currentSteppingEnabled;
END_SET
END_PROPERTY

{attribute 'hide'}
PROPERTY currentStepWidth : DINT
GET // PROTECTED
currentStepWidth := THIS^.stepStepWidth;
END_GET
SET
THIS^.stepStepWidth := currentStepWidth;
END_SET
END_PROPERTY

{attribute 'hide'}
PROPERTY currentStopRequestMode : CNM_CycleManagerInterfaces.StepStopRequestMode
GET // PROTECTED
currentStopRequestMode := THIS^.stepCurrentStopRequestMode;
END_GET
SET
THIS^.stepCurrentStopRequestMode := currentStopRequestMode;
END_SET
END_PROPERTY

(*

## Short summary
This property sets the maximum execution time for the current step. 
The cycle manager will go into the error step after the time elapsed.

.. <legal notes>

legal notes
=================
| SPDX-FileCopyrightText: © 2024 ekvip automation GmbH <info@ekvip.de>
| SPDX-License-Identifier: Apache-2.0
| For details check: Apache-2.0_

.. _Apache-2.0: https://www.apache.org/licenses/LICENSE-2.0

.. </legal notes>

*)
{attribute 'hide'}
PROPERTY currentTimeout : TIME
GET // PROTECTED
currentTimeout := THIS^.stepTimeOut;
END_GET
SET
THIS^.stepTimeOut := currentTimeout;
END_SET
END_PROPERTY

{attribute 'hide'}
PROPERTY currentTimeoutStep : DINT
GET // PROTECTED
IF(THIS^.stepTimeoutStep <> THIS^.defaultTimeoutStep OR THIS^.stepTimeoutStep <> THIS^.defaultErrorStep)THEN
	currentTimeoutStep := THIS^.stepTimeoutStep;	
ELSE
	currentTimeoutStep := THIS^.currentErrorStep;
END_IF
END_GET
SET
THIS^.stepTimeoutStep := currentTimeoutStep;
END_SET
END_PROPERTY

(*

## Short summary
This property stes the next step in case of an error after a step change.

.. <legal notes>

legal notes
=================
| SPDX-FileCopyrightText: © 2024 ekvip automation GmbH <info@ekvip.de>
| SPDX-License-Identifier: Apache-2.0
| For details check: Apache-2.0_

.. _Apache-2.0: https://www.apache.org/licenses/LICENSE-2.0

.. </legal notes>

*)

{attribute 'hide'}
PROPERTY defaultErrorStep : DINT
GET // PROTECTED
defaultErrorStep := THIS^.sequenceErrorStep;
END_GET
SET
THIS^.sequenceErrorStep := defaultErrorStep;
THIS^.currentErrorStep := defaultErrorStep;
END_SET
END_PROPERTY

(*

## Short summary
This property sets the default pause enabling state after a step change.

.. <legal notes>

legal notes
=================
| SPDX-FileCopyrightText: © 2024 ekvip automation GmbH <info@ekvip.de>
| SPDX-License-Identifier: Apache-2.0
| For details check: Apache-2.0_

.. _Apache-2.0: https://www.apache.org/licenses/LICENSE-2.0

.. </legal notes>

*)

{attribute 'hide'}
PROPERTY defaultPauseEnabled : BOOL
GET // PROTECTED
defaultPauseEnabled := THIS^.sequencePauseEnabled;
END_GET
SET
THIS^.sequencePauseEnabled := defaultPauseEnabled;
THIS^.currentPauseEnabled := defaultPauseEnabled;
END_SET
END_PROPERTY

(*

## Short summary
Specifies whether the SUCCESS step of the state machine can be skipped when the transition condition to SUCCESS is already fulfilled.

When set to false, the state machine immediately returns SUCCESS as soon as the transition condition to the SUCCESS state is met, 
without executing the dedicated SUCCESS step. This optimization can save one execution cycle per state machine invocation, which is 
especially beneficial in nested or complex state machine structures.

When set to true, the SUCCESS step will always be executed at least once before the state machine returns SUCCESS. This is required 
in cases where the SUCCESS step performs essential actions (e.g., resetting outputs, logging, or cleanup).

The default value is false.

Use Case:
Use false when the SUCCESS step has no functional side effects and skipping it can improve performance.
Use true when the SUCCESS step contains logic that must be executed explicitly.

.. <legal notes>

legal notes
=================
| SPDX-FileCopyrightText: © 2025 ekvip automation GmbH <info@ekvip.de>
| SPDX-License-Identifier: Apache-2.0
| For details check: Apache-2.0_

.. _Apache-2.0: https://www.apache.org/licenses/LICENSE-2.0

.. </legal notes>

*)

PROPERTY defaultRequireSuccessStep : BOOL
GET
defaultRequireSuccessStep := THIS^.sequenceRequireSuccessStep;
END_GET
SET
THIS^.sequenceRequireSuccessStep := defaultRequireSuccessStep;
END_SET
END_PROPERTY

(*

## Short summary
This property sets the default stepping mode configuration after a step change.

.. <legal notes>

legal notes
=================
| SPDX-FileCopyrightText: © 2024 ekvip automation GmbH <info@ekvip.de>
| SPDX-License-Identifier: Apache-2.0
| For details check: Apache-2.0_

.. _Apache-2.0: https://www.apache.org/licenses/LICENSE-2.0

.. </legal notes>

*)

{attribute 'hide'}
PROPERTY defaultSteppingEnabled : BOOL
GET // PROTECTED
defaultSteppingEnabled := THIS^.sequenceSteppingEnabled;
END_GET
SET
THIS^.sequenceSteppingEnabled := defaultSteppingEnabled;
THIS^.currentSteppingEnabled := defaultSteppingEnabled;
END_SET
END_PROPERTY

(*

## Short summary
This property sets the default the step width.

.. <legal notes>

legal notes
=================
| SPDX-FileCopyrightText: © 2024 ekvip automation GmbH <info@ekvip.de>
| SPDX-License-Identifier: Apache-2.0
| For details check: Apache-2.0_

.. _Apache-2.0: https://www.apache.org/licenses/LICENSE-2.0

.. </legal notes>

*)

{attribute 'hide'}
PROPERTY defaultStepWidth : DINT
GET // PROTECTED
defaultStepWidth := THIS^.sequenceStepWidth;
END_GET
SET
THIS^.sequenceStepWidth := defaultStepWidth;
THIS^.currentStepWidth := defaultStepWidth;
END_SET
END_PROPERTY

(*

## Short summary
This property sets the default step mode configuration. 

.. <legal notes>

legal notes
=================
| SPDX-FileCopyrightText: © 2024 ekvip automation GmbH <info@ekvip.de>
| SPDX-License-Identifier: Apache-2.0
| For details check: Apache-2.0_

.. _Apache-2.0: https://www.apache.org/licenses/LICENSE-2.0

.. </legal notes>

*)

{attribute 'hide'}
PROPERTY defaultStopRequestMode : CNM_CycleManagerInterfaces.StepStopRequestMode
GET // PROTECTED
defaultStopRequestMode := THIS^.sequenceStopRequestMode;
END_GET
SET
THIS^.sequenceStopRequestMode := defaultStopRequestMode;
THIS^.currentStopRequestMode := defaultStopRequestMode;
END_SET
END_PROPERTY

(*

## Short summary
This property sets the maximum execution time for steps. 
The cycle manager will go into the timeoutStep after the time elapsed.

.. <legal notes>

legal notes
=================
| SPDX-FileCopyrightText: © 2024 ekvip automation GmbH <info@ekvip.de>
| SPDX-License-Identifier: Apache-2.0
| For details check: Apache-2.0_

.. _Apache-2.0: https://www.apache.org/licenses/LICENSE-2.0

.. </legal notes>

*)

{attribute 'hide'}
PROPERTY defaultTimeout : TIME
GET // PROTECTED
defaultTimeout := THIS^.sequenceTimeOut;
END_GET
SET
THIS^.sequenceTimeOut := defaultTimeout;
THIS^.currentTimeout := defaultTimeout;
END_SET
END_PROPERTY

(*

## Short summary
This property sets the default step that will be set if the current step reaches a timeout. 

.. <legal notes>

legal notes
=================
| SPDX-FileCopyrightText: © 2024 ekvip automation GmbH <info@ekvip.de>
| SPDX-License-Identifier: Apache-2.0
| For details check: Apache-2.0_

.. _Apache-2.0: https://www.apache.org/licenses/LICENSE-2.0

.. </legal notes>

*)

{attribute 'hide'}
PROPERTY defaultTimeoutStep : DINT
GET // PROTECTED
defaultTimeoutStep := THIS^.sequenceTimeoutStep;
END_GET
SET
THIS^.sequenceTimeoutStep := defaultTimeoutStep;
THIS^.currentTimeoutStep := defaultTimeoutStep;
END_SET
END_PROPERTY

(*

## Short summary
This method performs the given invoke only in the first cycle of the current step.

.. <legal notes>

legal notes
=================
| SPDX-FileCopyrightText: © 2024 ekvip automation GmbH <info@ekvip.de>
| SPDX-License-Identifier: Apache-2.0
| For details check: Apache-2.0_

.. _Apache-2.0: https://www.apache.org/licenses/LICENSE-2.0

.. </legal notes>


*)
METHOD enter
VAR_INPUT
	(* command to execute *)
	invoke	:CNM_CommandInterfaces.ISingleAttempt;
	(* step to proceed with in case of error *)
	errorStep	:DINT := CNM_ReturnTypes.DefaultSteps.STEP.ERROR;
END_VAR
THIS^.registeredEnter := TRUE;

RETURN (
	THIS^.executeStep 
	OR_ELSE THIS^.state <> CNM_ReturnTypes.SingleExecutionState.BUSY
);

IF (THIS^.isObjectNull(invoke) OR_ELSE (invoke.invoke() <> CNM_ReturnTypes.SingleExecutionResult.SUCCESS)) THEN
	THIS^.wasError := TRUE;
	THIS^.wasSuccess := FALSE;
	IF ((errorStep <> CNM_ReturnTypes.DefaultSteps.STEP.ERROR) 
		AND_THEN (errorStep <> THIS^.currentErrorStep)
	) THEN
		THIS^.currentErrorStep := errorStep;
	END_IF
END_IF
END_METHOD

(*

